SUBAPPLICATION Softkey_Aux_IXA_TO_Remote_WRITE_BG_OPC (* VT-SoftKey lesen ODER AUX-Zuweisung (Joystick) lesen ODER lokaler Web-Override (z.B. vt-ui-mirror auf demselben Modul) + Remote-OPC-UA-Write an Zielmodul + VT-Hintergrundfarbe (SoftKey UND AUX) aus Remote-Subscribe (generisch, ein Kanal, fuer Funktionen ohne lokalen physischen Ausgang - Bedienung sitzt auf STG1, Aktor auf einem Modul ohne eigene VT-Anbindung) *)
  (* Standard: 61499-2; Description: Copyright (c) 2026 Meisterschulen am Ostbahnhof This program and the accompanying materials are made available under the terms of the Eclipse Public License 2.0 which is available at https://www.eclipse.org/legal/epl-2.0/ SPDX-License-Identifier: EPL-2.0 *)
  (* Version 1.2, 2026-09-07, Franz Höpfinger, Meisterschulen am Ostbahnhof, In 2 wiederverwendbare Teilbausteine zerlegt: Softkey_Aux_IXA_TO_Remote_WRITE (Kommando) + AX_SUBSCRIBE_BG3_WEB_OPC (Status) - externe Schnittstelle unveraendert *)
  (* Version 1.1, 2026-09-07, Franz Höpfinger, Meisterschulen am Ostbahnhof, Lokalen Status-Republish (ID_STATUS_WEB, AX_SPLIT_2, STATUS_WEB_PUBLISH) fuer Web-Clients ergaenzt *)
  (* Version 1.0, 2026-09-06, franz, Meisterschulen am Ostbahnhof *)
  PACKAGE MyLib::sys;
  (* Documentation:
  SoftKey UND Aux → Remote-OPC-UA-Write mit Status-Feedback auf beiden (ein Kanal)
   Duennwandiger Wrapper, der Softkey_Aux_IXA_TO_Remote_WRITE (Kommando: SoftKey ODER Aux ODER lokaler Web-Override → Remote-Write) und AX_SUBSCRIBE_BG3_WEB_OPC (Status: Remote-Subscribe → Hintergrundfarbe auf SoftKey UND Aux + lokaler Web-Republish) nebeneinanderstellt. Beide Teilbausteine sind eigenstaendig wiederverwendbar - dieser Wrapper existiert nur, damit ein Aufrufer weiterhin eine einzige SubApp mit der bekannten Schnittstelle instanziieren kann.
   Wird nur ein SoftKey ohne Aux gebraucht, Softkey_IXA_TO_Remote_WRITE_BG_OPC verwenden.
  *)
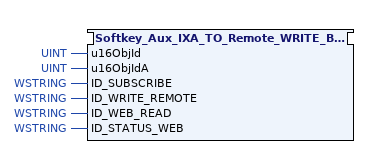
  VAR_INPUT
    u16ObjId : UINT; (* Object ID SoftKey/Hintergrund (VT) *)
    u16ObjIdA : UINT; (* Object ID AuxFunction2/Hintergrund (VT) *)
    ID_SUBSCRIBE : WSTRING; (* Remote-Subscribe-Adresse (Status/Farbe, ACTION=SUBSCRIBE) *)
    ID_WRITE_REMOTE : WSTRING; (* Remote-Write-Adresse zum Zielmodul (Befehl, ACTION=WRITE, CLIENT) *)
    ID_WEB_READ : WSTRING; (* Lokale Subscribe-Adresse fuer einen Web-Client (z.B. vt-ui-mirror) auf demselben Modul, ODER-verknuepft mit SoftKey und AUX *)
    ID_STATUS_WEB : WSTRING; (* Lokale Publish-Adresse (auf diesem Modul) fuer den vom Zielmodul zurueckgemeldeten Zustand - damit ein Web-Client (z.B. vt-ui-mirror) dieselbe Hintergrundfarbe wie das echte VT zeigen kann *)
  END_VAR
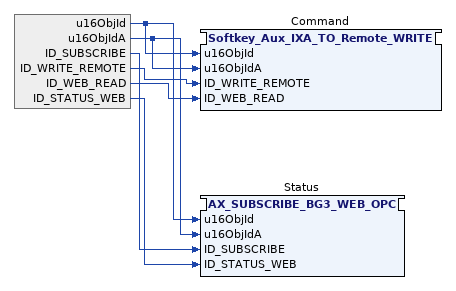
  SUBAPPS
    Command : MyLib::sys::Softkey_Aux_IXA_TO_Remote_WRITE;
    Status : MyLib::sys::AX_SUBSCRIBE_BG3_WEB_OPC;
  END_SUBAPPS
  DATA_CONNECTIONS
    u16ObjId TO Command.u16ObjId;
    u16ObjIdA TO Command.u16ObjIdA;
    ID_WRITE_REMOTE TO Command.ID_WRITE_REMOTE;
    ID_WEB_READ TO Command.ID_WEB_READ;
    u16ObjId TO Status.u16ObjId;
    u16ObjIdA TO Status.u16ObjIdA;
    ID_SUBSCRIBE TO Status.ID_SUBSCRIBE;
    ID_STATUS_WEB TO Status.ID_STATUS_WEB;
  END_CONNECTIONS
END_SUBAPPLICATION
